PROGRAM MAIN
VAR
	n_cnt_1 : UINT;
	n_cnt_2 : UINT;
	n_cnt_3 : UINT;
	
	ton_1 : TON := (PT := T#0.2S);
	ton_2 : TON := (PT := T#0.5S);
	ton_3 : TON := (PT := T#1S);
END_VAR

ton_1(IN := NOT ton_1.Q);
ton_2(IN := NOT ton_2.Q);
ton_3(IN := NOT ton_3.Q);

IF ton_1.Q THEN
	n_cnt_1 := n_cnt_1 + 1;
END_IF

IF ton_2.Q THEN
	n_cnt_2 := n_cnt_2 + 1;
END_IF

IF ton_3.Q THEN
	n_cnt_3 := n_cnt_3 + 1;
END_IF

END_PROGRAM

(* stored: Version 1.1.0.1, ProductVersion 3.1.4024.12
   POU MAIN: Id {245be3d9-2e3c-4a56-ab1d-124f45dc2728}, SpecialFunc None *)
